// TIA Portal V17 export
// export: Created 2021-12-03T08:12:56.6232568Z, ExportSetting WithDefaults, DisplayName Totally Integrated Automation Portal, DisplayVersion V17, DisplayName TIA Portal Openness, DisplayVersion V17, DisplayName TIA Portal Version Control Interface, DisplayVersion V17, DisplayName STEP 7 Professional, DisplayVersion V17, DisplayName STEP 7 Safety, DisplayVersion V17, DisplayName WinCC Advanced, DisplayVersion V17
DATA_BLOCK "DBI_GnrlFunc"   // DB2
VERSION : 0.1
// stored: AutoNumber true, InstanceOfName FB_GnrlFunc, InstanceOfType FB
"FB_GnrlFunc"
   // VAR RETAIN
   //    AxSR : Struct
   //       SrvcMd : Bool;
   //    END_STRUCT;
   // END_VAR
BEGIN
END_DATA_BLOCK
